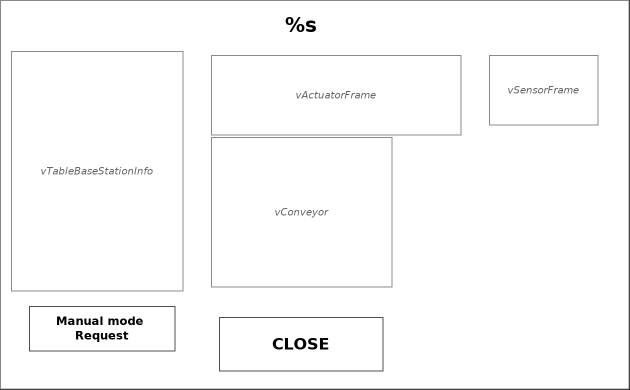
VISUALIZATION vTableUnoadingDetail  // 630x390
VAR_IN_OUT
	fbStation:FB_UnloadingStation;
	fbTableControl: FB_TableControl;
END_VAR
    Rectangle (0,0 630x390)
    Frame (11,51 172x240)
        shows vTableBaseStationInfo(fbStation := fbStation)
    Rectangle (219,317 164x54), "CLOSE"
        OnMouseDown: execute { fbTableControl.stHMI.iDialogNumber:=0; }
    Rectangle (226,10 150x30), "%s", text variable: fbStation.sStationName
    Frame (211,55 250x80)
        shows vActuatorFrame(iTextIndex1 := 4, iTextIndex2 := 5, fbActuator := fbStation.fbUnloadingActuator)
    Frame (489,55 109x70)
        shows vSensorFrame(iNameIndex := 1, fbSensor := fbStation.fbUnloadingSensor)
    Frame (211,137 181x150)
        shows vConveyor(iNameIndex := 5, fbConveyor := fbStation.fbConveyor)
    Rectangle (29,306 146x45), "Manual mode Request", colour toggle: fbStation.bManualModeRequest
        toggle fbStation.bManualModeRequest
END_VISUALIZATION

(* stored: Version 1.1.0.1, ProductVersion 3.1.4024.15
   Visu vTableUnoadingDetail: Id {daae760d-5af5-47cb-be83-3a2fa5ed4b32} *)
